Staubli VAL3: network.pjx

--- network.pjx ---
Parameters version=s7.11.2 stackSize=5000 millimeterUnit=true
Program file=start.pgx
Program file=stop.pgx
Data file=network.dtx

--- network.dtx ---
bool convnum = true
bool hasmsg
bool isx
bool isy = true
mdesc mNomSpeed
mdesc speed = {accel=9, vel=30, decel=9}
num cont
num divmsg = 5
num endmsg = 11
num gstart
num msg[32]
  [1] = 88
  [2] = 50
  [3] = 53
  [4] = 49
  [5] = 89
  [6] = 45
  [7] = 49
  [8] = 54
  [9] = 55
  [10] = 69
  [11] = 69
  [12] = 69
  [13] = 57
  [14] = 69
num xxx = 251
num yyy = -167
pointRs a = {x=407.52, y=-8.68, z=5.9, rx=-180, ry=-1.455991e-32, rz=-0.24, fatherId=world[0]}
pointRs home = {x=407.53, y=-8.71, z=140.1, rx=-180, ry=-1.412482e-32, rz=-0.23, fatherId=world[0]}
pointRs photo = {x=400, y=375, z=180, rx=-180, fatherId=world[0]}
sio input = {link=Socket\staubli}
string axxx = "251"
string ayyy = "-167"
string endchr = "E"
string message[32]
  [0] = "251-167"
  [1] = "M"
  [2] = "S"
  [3] = "G"
string split = "/"
tool garra = {x=20.5, y=13.05, z=13.77, fatherId=flange[0], ioLink=valve1}

--- start.pgx ---
program start()
begin
  // start
  enablePower()
  delay(0.9)
  movel(photo,garra,speed)
  waitEndMove()

  // worker
  while true
    // clear states and get message -> message: GXxxxYyyyDdE
      // X: x position
      // Y: y position
      // D: destination, is an integer value, with index of the points of cradle
    clearBuffer(input)
    cont=0
    sioGet(input,msg)
    hasmsg=chr(msg[0])=="G"
    // if has a valid message
    if hasmsg
      //clear worker states
      axxx=""
      ayyy=""
      message=""
      isy=false
      isx=false
      hasmsg=false
      cont=0
      while cont<31
        switch chr(msg[cont+1])
          case "E"
            cont=31
          break
          case "X"
            isx=true
            isy=false
          break
          case "Y"
            isx=false
            isy=true
          break
          default
            if isx
              axxx=axxx+chr(msg[cont+1])
            else
              ayyy=ayyy+chr(msg[cont+1])
            endIf
            message=message+chr(msg[cont+1])
          break
        endSwitch
        cont=cont+1
      endWhile

      //clear worker states
      cont=0
      msg=0

      // move to position
      toNum(axxx,xxx,convnum)
      toNum(ayyy,yyy,convnum)
      //move to home, then to position
      movej(home,garra,speed)
      waitEndMove()
      // [PICK]
      //move to position of the message
      movel(appro(home,{yyy,xxx,10,0,0,0}),garra,speed) //todo: cadastrar altura de approuch e pick
      waitEndMove()
      //get block : atual -> mover para baixo
      movel(appro({yyy,xxx,0,0,0,0},{0,0,heigth_pick,0,0,0}),garra,speed) // todo: cadastrar altura de pick
      waitEndMove()
      // ACTION: active gripper
      //atual -> mover para cima
      movel(appro({yyy,xxx,0,0,0,0}, {0,0,heigth_app,0,0,0}),garra,speed) // move to approuch again, after pick objetc
      waitEndMove()

      // [PLACE]
      //move to destination
      toNum(message,dest,convnum)
      movel(appro(home,cradle_appr[dest]),garra,speed)
      waitEndMove()
      movel(appro(cradle_appr[dest], {0,0,heigth_pick,0,0,0}),garra,speed) // move to approuch again, after pick objetc
      waitEndMove()
      // ACTION: active gripper
      movel(appro(cradle_appr[dest], {0,0,heigth_app,0,0,0}),garra,speed) // move to approuch again, after pick objetc
      waitEndMove()
      //move to home to end
      movej(home,garra,speed)
      waitEndMove()



    else
    endIf
    //
  endWhile
  //
  //
end
